FUNCTION BP_TO_IO : ST_BeamParams_IO
VAR_INPUT
    BP : ST_BeamParams;
END_VAR
VAR
    idx : UINT := 0;
END_VAR


FOR idx := 1 TO PMPS_GVL.AUX_ATTENUATORS DO
    BP_TO_IO.astAttenuators[idx] := ATT_TO_IO(BP.astAttenuators[idx]);
END_FOR

BP_TO_IO.aStoppers := BP.aStoppers;
BP_TO_IO.fAtt := BP.fAtt;
BP_TO_IO.fPP_mJ := BP.fPP_mJ;
BP_TO_IO.nCohortInt := ULINT_TO_UDINT(BP.nCohortInt);
BP_TO_IO.neVRange := BP.neVRange;
BP_TO_IO.nRate := BP.nRate;
BP_TO_IO.xValid := BP.xValid;
BP_TO_IO.xValidToggle := BP.xValidToggle;

END_FUNCTION

(* stored: Version 1.1.0.1, ProductVersion 3.1.4022.18
   POU BP_TO_IO: Id {99655e6a-0c9e-47fa-acc0-f263faf87725}, SpecialFunc None *)
